# EPICS substitutions: ek9000App/Db/EL4001.substitutions
file EL4001.template
{       pattern
        {
                TERMINAL,

        }
        {
        }
}
